FUNCTION_BLOCK FB_Vec3 IMPLEMENTS I_Vec3
VAR_INPUT
END_VAR
VAR_OUTPUT
END_VAR
VAR
END_VAR


{warning 'Add method implementation '}
METHOD AddVec3 : I_Vec3
VAR_INPUT
    iVec3	: I_Vec3;
END_VAR
END_METHOD


{warning 'Add method implementation '}
METHOD CrossVec3 : I_Vec3
VAR_INPUT
    iVec3	: I_Vec3;
END_VAR
END_METHOD


{warning 'Add method implementation '}
METHOD DotVec3 : LREAL
VAR_INPUT
    iVec3	: I_Vec3;
END_VAR
END_METHOD


{warning 'Add method implementation '}
METHOD GetMag : LREAL
END_METHOD


{warning 'Add method implementation '}
METHOD GetNorm : I_Vec3
END_METHOD


{warning 'Add method implementation '}
METHOD ToString : STRING
END_METHOD


{warning 'Add property implementation'}
PROPERTY x : LREAL
GET
END_GET
END_PROPERTY


{warning 'Add property implementation'}
PROPERTY y : LREAL
GET
END_GET
END_PROPERTY


{warning 'Add property implementation'}
PROPERTY z : LREAL
GET
END_GET
END_PROPERTY

END_FUNCTION_BLOCK

(* stored: Version 1.1.0.1
   POU FB_Vec3: Id {c09dfe87-9fa9-4800-966a-c9fa2f01d9b6}, SpecialFunc None
   Method AddVec3: Id {ef14f849-964d-41c6-b93c-957ccd6460f6}
   Method CrossVec3: Id {61d300cc-4420-46cd-b758-e15093cacda1}
   Method DotVec3: Id {96055ecf-9626-4c41-8898-10ce4518584b}
   Method GetMag: Id {9a7fc225-e930-434a-aa42-0d79876ee438}
   Method GetNorm: Id {29814131-65a5-4ed7-b948-b70d7762daf7}
   Method ToString: Id {c35ca60f-311e-4b45-99f0-9b9fae4ea9dd}
   Property x: Id {d1132b1f-8d78-4d71-868f-4b5ca1d3abf5}
   Get Get: Id {f7878e76-22eb-42c2-97b3-b87e70fce12d}
   Property y: Id {9bbfc62e-5928-4dd9-9c9f-a12c08bc7ea3}
   Get Get: Id {8be5870a-3987-4750-b25a-35c6debc60c5}
   Property z: Id {668d9da2-5ed3-4ecb-9b12-26772daecde7}
   Get Get: Id {51c53bf0-f603-4526-af72-51056970282d} *)
